FUNCTION_BLOCK CsvByteDocumentWriter IMPLEMENTS I_CsvDocument, I_CsvRecord
VAR
	
	byteBuffer : I_Buffer;
	fieldStyle : (NEW_FIELD,NEXT_FIELD) := NEW_FIELD;
	_useQuotes : BOOL := TRUE;
	_fieldCount : UDINT;
	_recordCount : UDINT;
	_fieldDivider : BYTE := F_ToASC(';');
	_recordEnd : STRING := '$0D$0A';
	quoteMark : BYTE := F_ToASC('"'); 
	
END_VAR

METHOD PUBLIC AddBool : I_CsvRecord;
VAR_IN_OUT
	Field : BOOL;
END_VAR
BeforeAddFieldOperations();
byteBuffer.AddBoolToBuffer(Field);
AfterAddFieldOperations();
AddBool := THIS^;
END_METHOD

METHOD PUBLIC AddBoolLiteral : I_CsvRecord;
VAR_INPUT
	Field : BOOL;
END_VAR
BeforeAddFieldOperations();
byteBuffer.AddBoolToBuffer(Field);
AfterAddFieldOperations();
AddBoolLiteral := THIS^;
END_METHOD

METHOD PROTECTED AddFieldDividerToBuffer
byteBuffer.AddCharToBuffer(_fieldDivider);
END_METHOD

METHOD PUBLIC AddInt : I_CsvRecord;
VAR_IN_OUT
	Field : INT;
END_VAR
BeforeAddFieldOperations();
byteBuffer.AddIntToBuffer(Field);
AfterAddFieldOperations();
AddInt := THIS^;
END_METHOD

METHOD PUBLIC AddIntLiteral : I_CsvRecord;
VAR_INPUT
	Field : INT;
END_VAR
BeforeAddFieldOperations();
byteBuffer.AddIntToBuffer(Field);
AfterAddFieldOperations();
AddIntLiteral := THIS^;
END_METHOD

METHOD PROTECTED AddQuoteToBuffer
byteBuffer.AddCharToBuffer(quoteMark);
END_METHOD

METHOD PROTECTED AddRecordEndCharactersToBuffer
byteBuffer.AddStringToBuffer(_recordEnd);
END_METHOD

METHOD PUBLIC AddString : I_CsvRecord;
VAR_IN_OUT
	stringToWrite : STRING;
END_VAR
BeforeAddFieldOperations();
byteBuffer.AddStringToBuffer(stringToWrite);
AfterAddFieldOperations();
AddString := THIS^;
END_METHOD

METHOD PUBLIC AddStringLiteral : I_CsvRecord;
VAR_INPUT
	stringToWrite : STRING;
END_VAR
BeforeAddFieldOperations();
byteBuffer.AddStringToBuffer(stringToWrite);
AfterAddFieldOperations();
AddStringLiteral := THIS^;
END_METHOD

METHOD AddULint : I_CsvRecord
VAR_IN_OUT
	Field	: ULINT;
END_VAR
BeforeAddFieldOperations();
byteBuffer.AddULintToBuffer(Field);
AfterAddFieldOperations();
AddULint := THIS^;
END_METHOD

METHOD AddULintLiteral : I_CsvRecord
VAR_INPUT
	Field	: ULINT;
END_VAR
BeforeAddFieldOperations();
byteBuffer.AddULintToBuffer(Field);
AfterAddFieldOperations();
AddULintLiteral := THIS^;
END_METHOD

METHOD PROTECTED AfterAddFieldOperations
IF _useQuotes THEN
	AddQuoteToBuffer();
END_IF

fieldStyle := NEXT_FIELD;
_fieldCount := _fieldCount + 1;
END_METHOD

METHOD PROTECTED BeforeAddFieldOperations
IF fieldStyle = NEXT_FIELD THEN
	AddFieldDividerToBuffer();
END_IF

IF _useQuotes THEN
	AddQuoteToBuffer();
END_IF
END_METHOD

METHOD PUBLIC EndRecord : I_CsvDocument;
AddRecordEndCharactersToBuffer();
_recordCount := _recordCount + 1;
EndRecord := THIS^;
END_METHOD

METHOD FB_init : BOOL
VAR_INPUT
	bInitRetains : BOOL; // if TRUE, the retain variables are initialized (warm start / cold start)
	bInCopyCode : BOOL;  // if TRUE, the instance afterwards gets moved into the copy code (online change)
	ByteBuffer : I_Buffer;
END_VAR
THIS^.byteBuffer := ByteBuffer;
END_METHOD

PROPERTY PUBLIC FieldCount : UDINT
GET
FieldCount := _fieldCount;
END_GET
END_PROPERTY

PROPERTY PUBLIC FieldDivider : BYTE
GET
FieldDivider := _fieldDivider;
END_GET
SET
_fieldDivider := FieldDivider;
END_SET
END_PROPERTY

PROPERTY PUBLIC IsFull : BOOL
GET
IsFull := byteBuffer.Remaining = 0;
END_GET
END_PROPERTY

PROPERTY PUBLIC RecordCount : UDINT
GET
RecordCount := _recordCount;
END_GET
END_PROPERTY

METHOD Reset
VAR_INPUT
END_VAR
byteBuffer.Reset();
_recordCount := 0;
_fieldCount := 0;
END_METHOD

METHOD PUBLIC StartRecord : reference to CsvByteDocumentWriter//I_CsvRecordWriter
VAR_INPUT
END_VAR
fieldStyle := NEW_FIELD;
StartRecord ref= this^;
END_METHOD

METHOD PUBLIC UpdateBuffer
VAR_INPUT
	Buffer : POINTER TO BYTE;
	BufferSize : UDINT;
END_VAR
END_METHOD

PROPERTY PUBLIC UseQuotes : BOOL
GET
UseQuotes := _useQuotes;
END_GET
SET
_useQuotes := UseQuotes;
END_SET
END_PROPERTY

END_FUNCTION_BLOCK

(* stored: Version 1.1.0.1, ProductVersion 3.1.4024.4
   POU CsvByteDocumentWriter: Id {fb521214-c9d1-42fc-87a9-31391909d3df}, SpecialFunc None
   Folder Constructor: Id {bafcd508-3932-4f44-990b-4d1ac49d8171}
   Folder Private: Id {e4076296-8d10-4254-90d3-74d8385b5d87}
   Folder Properties: Id {52acf36a-f1da-41a8-8b5b-f746b5b3ce15}
   Method AddBool: Id {c8324f9f-d703-4093-a9e8-2270acd0312e}
   Method AddBoolLiteral: Id {a0756402-09de-424a-958c-8035b9a49809}
   Method AddFieldDividerToBuffer: Id {d49b5001-57f1-472a-8e22-8cd59cc089ac}
   Method AddInt: Id {7510350b-74c2-4364-9e17-e500b4437411}
   Method AddIntLiteral: Id {3db738bd-7aae-4d74-aad9-ac9a7c8578a4}
   Method AddQuoteToBuffer: Id {f5432f9a-23a6-456e-a6cc-08c440c62116}
   Method AddRecordEndCharactersToBuffer: Id {f52cd7ac-5d45-413a-97f5-50cdf368bceb}
   Method AddString: Id {4c39018d-acbd-47f3-88cc-a7906d7184b2}
   Method AddStringLiteral: Id {c11fa6cd-5757-42d6-a2c0-d2edee7189d8}
   Method AddULint: Id {02982d7e-e453-4377-8f35-adafb7ab4fc0}
   Method AddULintLiteral: Id {83fb0f0e-9941-4b25-907f-0796bb596871}
   Method AfterAddFieldOperations: Id {3fcf919f-9762-42a6-a5ab-708f62b01355}
   Method BeforeAddFieldOperations: Id {5d7fa340-4f23-4e43-8dd7-3dd989c5cf14}
   Method EndRecord: Id {810018e0-cf29-4469-a7da-7d5d4ea4cf61}
   Method FB_init: Id {d76499c9-18f2-4c02-b05f-c94cbda18ab1}
   Property FieldCount: Id {1ed7f8dd-dbd6-4408-a3e2-f98e86bd24ca}
   Get Get: Id {dade60af-6a6e-400a-9a20-142bd25d52e9}
   Property FieldDivider: Id {644c17bb-67d1-47cc-b79c-c8f2f2ff0fae}
   Get Get: Id {c6af6698-dd5e-49ee-8c9d-d925f47c8ea7}
   Set Set: Id {ab389e68-2935-4d92-a66f-c6163edb0093}
   Property IsFull: Id {54550429-0f28-4476-aad0-07497278423a}
   Get Get: Id {8e41b8f6-eda1-4113-a151-f6359a4116d6}
   Property RecordCount: Id {67502d15-391c-43e7-8ac8-f52f5ff47c1f}
   Get Get: Id {984cf197-c40a-4fdd-9fb7-254335d077b0}
   Method Reset: Id {3686be07-a445-4742-b565-e1898ee45ccc}
   Method StartRecord: Id {718c1d6a-763a-4544-9e14-58056349b870}
   Method UpdateBuffer: Id {db3a0aff-1fe3-4bef-8b1a-1ed869678b8d}
   Property UseQuotes: Id {e7602b62-b756-4a38-91a6-4a6ebb9f5965}
   Get Get: Id {026a1190-b91d-415a-9c9a-7d1752e97a48}
   Set Set: Id {c2133992-63ab-4111-b14c-b2cd0a00681b} *)
